PROGRAM PRG_TerminalMapping
VAR
    uiIndexPositionCode : UINT;
END_VAR

METHOD PUBLIC ReadInputs
(*
======================================================================================================================
 Terminal 4 | EL1918
======================================================================================================================
*)
GVL_IO.stInputs.bEmergencyStopChannel1 	:= GVL_EtherCAT.stTerm4_EL1918.iEL1918_Ch1;
GVL_IO.stInputs.bEmergencyStopChannel2 	:= GVL_EtherCAT.stTerm4_EL1918.iEL1918_Ch2;
// Reset is exported by TwinSAFE. Use the validated alias rather than
// reconstructing the operator Reset from a raw safety-terminal channel.
GVL_IO.stInputs.bResetButton 			:= GVL_Safety.bResetButtonPressed;
GVL_IO.stInputs.bMainDoorChannel1 		:= GVL_EtherCAT.stTerm4_EL1918.iEL1918_Ch4;
GVL_IO.stInputs.bMainDoorChannel2 		:= GVL_EtherCAT.stTerm4_EL1918.iEL1918_Ch5;
GVL_IO.stInputs.bMainDoorFeedback 		:= GVL_EtherCAT.stTerm4_EL1918.iEL1918_Ch6;
GVL_IO.stInputs.bMs6FeedbackOk 			:= GVL_EtherCAT.stTerm4_EL1918.iEL1918_Ch7;
GVL_IO.stInputs.bAirExhausted 			:= GVL_EtherCAT.stTerm4_EL1918.iEL1918_Ch8;

(*
======================================================================================================================
 Terminal 5 | EL1918
======================================================================================================================
*)
GVL_IO.stInputs.bTouchButtonLeft 		:= GVL_EtherCAT.stTerm5_EL1918.iEL1918_Ch3;
GVL_IO.stInputs.bTouchButtonRight 		:= GVL_EtherCAT.stTerm5_EL1918.iEL1918_Ch4;
GVL_IO.stInputs.bRightFlapChannel1 		:= GVL_EtherCAT.stTerm5_EL1918.iEL1918_Ch5;
GVL_IO.stInputs.bRightFlapChannel2 		:= GVL_EtherCAT.stTerm5_EL1918.iEL1918_Ch6;
GVL_IO.stInputs.bLeftFlapChannel1 		:= GVL_EtherCAT.stTerm5_EL1918.iEL1918_Ch7;
GVL_IO.stInputs.bLeftFlapChannel2 		:= GVL_EtherCAT.stTerm5_EL1918.iEL1918_Ch8;

(*
======================================================================================================================
 Terminal 7 | EL1809
======================================================================================================================
*)
GVL_IO.stInputs.bStartButton 				:= GVL_EtherCAT.stTerm7_EL1809.iEL1809_Ch1;
GVL_IO.stInputs.bStopButton 				:= NOT GVL_EtherCAT.stTerm7_EL1809.iEL1809_Ch2;
GVL_IO.stInputs.bUp24VPowerSupplyOk 		:= GVL_EtherCAT.stTerm7_EL1809.iEL1809_Ch3;
GVL_IO.stInputs.bUs24VPowerSupplyOk 		:= GVL_EtherCAT.stTerm7_EL1809.iEL1809_Ch4;
GVL_IO.stInputs.b48VPowerSupplyOk 			:= GVL_EtherCAT.stTerm7_EL1809.iEL1809_Ch5;
GVL_IO.stInputs.bIndexPositionSensor1 		:= GVL_EtherCAT.stTerm7_EL1809.iEL1809_Ch6;
GVL_IO.stInputs.bIndexPositionSensor2 		:= GVL_EtherCAT.stTerm7_EL1809.iEL1809_Ch7;
GVL_IO.stInputs.bIndexPositionSensor3 		:= GVL_EtherCAT.stTerm7_EL1809.iEL1809_Ch8;
GVL_IO.stInputs.bIndexCompletedSensor 		:= GVL_EtherCAT.stTerm7_EL1809.iEL1809_Ch9;
GVL_IO.stInputs.bIndexLocked 				:= GVL_EtherCAT.stTerm7_EL1809.iEL1809_Ch10;
GVL_IO.stInputs.bIndexReady 				:= GVL_EtherCAT.stTerm7_EL1809.iEL1809_Ch11;
GVL_IO.stInputs.bLoadingStationEaglePresent := GVL_EtherCAT.stTerm7_EL1809.iEL1809_Ch12;
GVL_IO.stInputs.bRejectChutePartPresent 	:= GVL_EtherCAT.stTerm7_EL1809.iEL1809_Ch13;
GVL_IO.stInputs.bHeatStakeEaglePresent 		:= GVL_EtherCAT.stTerm7_EL1809.iEL1809_Ch14;
GVL_IO.stInputs.bLoadingStationPbupPresent	:= GVL_EtherCAT.stTerm7_EL1809.iEL1809_Ch15;
GVL_IO.stInputs.bPbupMagnetPresent 			:= GVL_EtherCAT.stTerm7_EL1809.iEL1809_Ch16;

(*
======================================================================================================================
 INDEX Position
======================================================================================================================
*)
uiIndexPositionCode := 0;

IF GVL_IO.stInputs.bIndexPositionSensor1 THEN 
	uiIndexPositionCode := uiIndexPositionCode + 1; 
END_IF

IF GVL_IO.stInputs.bIndexPositionSensor2 THEN 
	uiIndexPositionCode := uiIndexPositionCode + 2; 
END_IF

IF GVL_IO.stInputs.bIndexPositionSensor3 THEN 
	uiIndexPositionCode := uiIndexPositionCode + 4; 
END_IF

IF GVL_IO.stInputs.bIndexLocked THEN 
	GVL_IO.stInputs.eIndexPosition := UINT_TO_E_TablePosition(uiIndexPositionCode);
ELSE 
	GVL_IO.stInputs.eIndexPosition := E_TablePosition.Unknown; 
END_IF

(*
======================================================================================================================
 Terminal 8 | EL1809
======================================================================================================================
*)

GVL_IO.stInputs.bStation1SupportRetracted := FALSE; // Retired compatibility field; EL1809 Ch1/Ch2 reserved.
GVL_IO.stInputs.bStation1SupportExtended := FALSE; // Retired compatibility field; EL1809 Ch1/Ch2 reserved.
GVL_IO.stInputs.bStation2SupportRetracted 		:= GVL_EtherCAT.stTerm8_EL1809.iEL1809_Ch3;
GVL_IO.stInputs.bStation2SupportExtended 		:= GVL_EtherCAT.stTerm8_EL1809.iEL1809_Ch4;
GVL_IO.stInputs.bStation3SupportRetracted := FALSE; // Retired compatibility field; raw terminal stays diagnostic-only.
GVL_IO.stInputs.bStation3SupportExtended := FALSE; // Retired compatibility field; raw terminal stays diagnostic-only.
GVL_IO.stInputs.bHorizontalMiniSlideRetracted 	:= GVL_EtherCAT.stTerm8_EL1809.iEL1809_Ch7;
GVL_IO.stInputs.bHorizontalMiniSlideExtended 	:= GVL_EtherCAT.stTerm8_EL1809.iEL1809_Ch8;
GVL_IO.stInputs.bVerticalMiniSlideExtended		:= GVL_EtherCAT.stTerm8_EL1809.iEL1809_Ch9;
GVL_IO.stInputs.bVerticalMiniSlideRetracted 	:= GVL_EtherCAT.stTerm8_EL1809.iEL1809_Ch10;
GVL_IO.stInputs.bIntermediateModuleRetracted := FALSE; // Retired compatibility field; raw terminal stays diagnostic-only.
GVL_IO.stInputs.bIntermediateModuleExtended := FALSE; // Retired compatibility field; raw terminal stays diagnostic-only.
GVL_IO.stInputs.bRotaryGripperOpened 			:= GVL_EtherCAT.stTerm8_EL1809.iEL1809_Ch13;
GVL_IO.stInputs.bRotaryGripperClosed 			:= GVL_EtherCAT.stTerm8_EL1809.iEL1809_Ch14;
GVL_IO.stInputs.bRotaryGripperPick0             := GVL_EtherCAT.stTerm8_EL1809.iEL1809_Ch16;
GVL_IO.stInputs.bRotaryGripperPlace180          := GVL_EtherCAT.stTerm8_EL1809.iEL1809_Ch15;

(*
======================================================================================================================
 Terminal 19 | EL1809
======================================================================================================================
*)

// Provisional operator PBUP presence; move this mapping when the final terminal is assigned.
//GVL_IO.stInputs.bLoadingStationPbupPresent 	:= GVL_EtherCAT.stTerm19_EL1809.iEL1809_Ch1;
GVL_IO.stInputs.bPatchOpticalLeft 			:= GVL_EtherCAT.stTerm19_EL1809.iEL1809_Ch5;
GVL_IO.stInputs.bPatchOpticalRight 			:= GVL_EtherCAT.stTerm19_EL1809.iEL1809_Ch6;
GVL_IO.stInputs.bHeatStakeHeadUp   			:= GVL_EtherCAT.stTerm19_EL1809.iEL1809_Ch7;
GVL_IO.stInputs.bHeatStakeHeadDown 			:= GVL_EtherCAT.stTerm19_EL1809.iEL1809_Ch8;
GVL_IO.stInputs.bMembraneTransferRetracted 	:= GVL_EtherCAT.stTerm19_EL1809.iEL1809_Ch9;
GVL_IO.stInputs.bMembraneTransferExtended 	:= GVL_EtherCAT.stTerm19_EL1809.iEL1809_Ch10;
GVL_IO.stInputs.bMiddleRockerDown 			:= GVL_EtherCAT.stTerm19_EL1809.iEL1809_Ch11;
GVL_IO.stInputs.bMiddleRockerUp 			:= GVL_EtherCAT.stTerm19_EL1809.iEL1809_Ch12;
GVL_IO.stInputs.bBottomRockerDown 			:= GVL_EtherCAT.stTerm19_EL1809.iEL1809_Ch13;
GVL_IO.stInputs.bBottomRockerUp 			:= GVL_EtherCAT.stTerm19_EL1809.iEL1809_Ch14;
GVL_IO.stInputs.bTopRockerDown 				:= GVL_EtherCAT.stTerm19_EL1809.iEL1809_Ch15;
GVL_IO.stInputs.bTopRockerUp 				:= GVL_EtherCAT.stTerm19_EL1809.iEL1809_Ch16;

(*
======================================================================================================================
 Terminal 11 | EL3058
======================================================================================================================
*)
GVL_IO.stInputs.uiMainAirPressureRaw 		 := GVL_EtherCAT.stTerm11_EL3058.iEL3058_Ch1;
GVL_IO.stInputs.uiPressureRegulatorActualRaw := GVL_EtherCAT.stTerm11_EL3058.iEL3058_Ch2;

(*
======================================================================================================================
 Terminal 20 | EL3314-0092 | Heat Stake Thermocouples
======================================================================================================================
*)
GVL_IO.stInputs.diHeatStakeTc1Raw := GVL_EtherCAT.stTerm21_EL3314.iEL3314_Ch1;
GVL_IO.stInputs.diHeatStakeTc2Raw := GVL_EtherCAT.stTerm21_EL3314.iEL3314_Ch2;
GVL_IO.stInputs.diHeatStakeTc3Raw := GVL_EtherCAT.stTerm21_EL3314.iEL3314_Ch3;

(*
======================================================================================================================
 SAFETY ALIAS Inputs
======================================================================================================================
*)
GVL_IO.stInputs.bSafetyOk 				:= GVL_Safety.bSafetyOk;
GVL_IO.stInputs.bTwoHandsSafe 			:= GVL_Safety.bTwoHandSafe;
GVL_IO.stInputs.bMainDoorClosed 		:= GVL_Safety.bMainDoorClosed;
GVL_IO.stInputs.bMainDoorLocked 		:= GVL_Safety.bMainDoorLocked;
GVL_IO.stInputs.bMainDoorUnsafe 		:= GVL_Safety.bMainDoorUnSafe;
GVL_IO.stInputs.bMainDoorDiagnosticOk 	:= GVL_Safety.bMainDoorDiagnosticOk;
END_METHOD

METHOD PUBLIC WriteOutputs
(*
======================================================================================================================
 SAFETY Alias Outputs
======================================================================================================================
*)
GVL_Safety.bSafetyRunRequest 					:= GVL_IO.stOutputs.bSafetyRunRequest;
GVL_Safety.bSafetyResetRequest 					:= GVL_IO.stOutputs.bSafetyResetRequest;
GVL_Safety.bSafetyErrorAcknowledgementRequest 	:= GVL_IO.stOutputs.bSafetyErrorAcknowledgementRequest;
GVL_Safety.bAirSupplyEnableRequest 				:= GVL_IO.stOutputs.bAirSupplyEnable;
GVL_Safety.bMainDoorLockRequest 				:= GVL_IO.stOutputs.bMainDoorLockRequest;

(*
======================================================================================================================
 Terminal 9 | EL2809
======================================================================================================================
*)
GVL_EtherCAT.stTerm9_EL2809.iEL2809_Ch1 := GVL_IO.stOutputs.bLedStart;
GVL_EtherCAT.stTerm9_EL2809.iEL2809_Ch2 := GVL_IO.stOutputs.bLedReset;

// Validated physical status-light mapping:
// Ch3 = RED status indicator (driven from machine FAIL)
// Ch4 = GREEN status indicator (driven from machine PASS)
GVL_EtherCAT.stTerm9_EL2809.iEL2809_Ch3 := GVL_IO.stOutputs.bStatusIndicatorRed;
GVL_EtherCAT.stTerm9_EL2809.iEL2809_Ch4 := GVL_IO.stOutputs.bStatusIndicatorGreen;

// Ch5 = internal cabinet/machine light
// Ch6 = operator/nest light
GVL_EtherCAT.stTerm9_EL2809.iEL2809_Ch5 := GVL_IO.stOutputs.bInternalLight;
GVL_EtherCAT.stTerm9_EL2809.iEL2809_Ch6 := GVL_IO.stOutputs.bNestLight;
// Monostable Heat Stake valve: TRUE = UP, FALSE = DOWN.
GVL_EtherCAT.stTerm9_EL2809.iEL2809_Ch7 := GVL_IO.stOutputs.bHeatStakeHeadUp;

(*
======================================================================================================================
 Terminal 13 | EL2502 | Heat Stake PWM Outputs
======================================================================================================================
*)
// IMPORTANT - VALIDATED PHYSICAL MAPPING.
// The heater channels are intentionally crossed relative to logical Heater 1 / Heater 2.
//
// EL2502 Ch1 physically drives logical Heater 2.
// EL2502 Ch2 physically drives logical Heater 1.
GVL_EtherCAT.stTerm13_EL2502.iEL2502_Ch1 := GVL_IO.stOutputs.uiHeatStakePwm2Raw;
GVL_EtherCAT.stTerm13_EL2502.iEL2502_Ch2 := GVL_IO.stOutputs.uiHeatStakePwm1Raw;

(*
======================================================================================================================
 Terminal 21 | EL4028 | VEAB Heat Stake Down Pressure
======================================================================================================================
*)
GVL_EtherCAT.stTerm20_EL4022.iEL4028_Ch1 := GVL_IO.stOutputs.iHeatStakePressureRaw;

(*
======================================================================================================================
 BOX 1 | Festo VABX EtherCAT manifold - Module 2
======================================================================================================================
*)

// Module2.Coil0 = Index Table A - rotate index
// Module2.Coil1 = Index Table B - return index cylinder to home
// Module2.Coil2 = RESERVED - removed Patch nest support UP
// Module2.Coil3 = RESERVED - removed Patch nest support DOWN
// Module2.Coil4 = Support UP   - Heat Stake Station
// Module2.Coil5 = Support DOWN - Heat Stake Station
// Module2.Coil6 = Support UP   - Vision Station
// Module2.Coil7 = Support DOWN - Vision Station
//
// Application naming:
// UP   = Extend
// DOWN = Retract
GVL_EtherCAT.stFestoModule2_VABX.bCoil0 := GVL_IO.stOutputs.bIndexRotatePortA;
GVL_EtherCAT.stFestoModule2_VABX.bCoil1 := GVL_IO.stOutputs.bIndexStopPortB;

GVL_EtherCAT.stFestoModule2_VABX.bCoil2 := FALSE; // Removed Patch nest support; keep valve OFF.
GVL_EtherCAT.stFestoModule2_VABX.bCoil3 := FALSE; // Reserved, not reassigned.

GVL_EtherCAT.stFestoModule2_VABX.bCoil4 := GVL_IO.stOutputs.bStation2SupportExtend;
GVL_EtherCAT.stFestoModule2_VABX.bCoil5 := GVL_IO.stOutputs.bStation2SupportRetract;

GVL_EtherCAT.stFestoModule2_VABX.bCoil6 := FALSE; // Removed Vision hardware: never energise.
GVL_EtherCAT.stFestoModule2_VABX.bCoil7 := FALSE; // Removed Vision hardware: never energise.

(*
======================================================================================================================
 BOX 1 | Festo VABX EtherCAT manifold - Module 3 | Vision Flipping
======================================================================================================================
*)
// Mapping confirmed from the commissioned GVL_EtherCAT / manifold layout.
// Coil0 = Horizontal slide BACK
// Coil1 = Horizontal slide FRONT
// Coil2 = Vertical cylinder UP
// Coil3 = Vertical cylinder DOWN
// Coil4 = Vertical cylinder limit OFF
// Coil5 = Vertical cylinder limit ON
// Coil6 = Grip CLOSE
// Coil7 = Grip OPEN
GVL_EtherCAT.stFestoModule3_VABX.bCoil0 := GVL_IO.stOutputs.bVisionHorizontalBack;
GVL_EtherCAT.stFestoModule3_VABX.bCoil1 := GVL_IO.stOutputs.bVisionHorizontalFront;
GVL_EtherCAT.stFestoModule3_VABX.bCoil2 := GVL_IO.stOutputs.bVisionVerticalUp;
GVL_EtherCAT.stFestoModule3_VABX.bCoil3 := GVL_IO.stOutputs.bVisionVerticalDown;
GVL_EtherCAT.stFestoModule3_VABX.bCoil4 := FALSE; // Removed Vision hardware: never energise.
GVL_EtherCAT.stFestoModule3_VABX.bCoil5 := FALSE; // Removed Vision hardware: never energise.
GVL_EtherCAT.stFestoModule3_VABX.bCoil6 := GVL_IO.stOutputs.bVisionGripOpen;
GVL_EtherCAT.stFestoModule3_VABX.bCoil7 := GVL_IO.stOutputs.bVisionGripClose;
(*
======================================================================================================================
 BOX 1 | Festo VABX EtherCAT manifold - Module 4 | Heat Stake Head
======================================================================================================================
*)
// Mapping confirmed from the commissioned GVL_EtherCAT / manifold layout.
// Coil0 = Vision gripper rotation 0Â° / PICK
// Coil1 = Vision gripper rotation 180Â° / PLACE
// Coil2 = Patch dispenser AIR
// Coil3 = Heat Stake head UNLOCK
// Coil4 = retired head DOWN output (always OFF)
// Coil5 = continuous pilot supply for the external head valve
// Coil6 = Patch vertical support DOWN
// Coil7 = Patch vertical support UP

GVL_EtherCAT.stFestoModule4_VABX.bCoil0 := GVL_IO.stOutputs.bVisionRotate0;
GVL_EtherCAT.stFestoModule4_VABX.bCoil1 := GVL_IO.stOutputs.bVisionRotate180;
GVL_EtherCAT.stFestoModule4_VABX.bCoil2 := GVL_IO.stOutputs.bPatchDispenserAir;
GVL_EtherCAT.stFestoModule4_VABX.bCoil3 := GVL_IO.stOutputs.bHeatStakeHeadUnlock;
GVL_EtherCAT.stFestoModule4_VABX.bCoil4 := FALSE; // Retired direction output.
GVL_EtherCAT.stFestoModule4_VABX.bCoil5 := TRUE; // Continuous pilot supply; reservoir supports retraction.
GVL_EtherCAT.stFestoModule4_VABX.bCoil6 := GVL_IO.stOutputs.bPatchVerticalDown;
GVL_EtherCAT.stFestoModule4_VABX.bCoil7 := GVL_IO.stOutputs.bPatchVerticalUp;
END_METHOD

END_PROGRAM

(* stored: Version 1.1.0.1, ProductVersion 3.1.4026.18
   POU PRG_TerminalMapping: Id {238243cb-7891-4569-b868-8787a9e2c958}, SpecialFunc None
   Method ReadInputs: Id {dd42962b-99a1-4f07-bcc4-f10d6e3158eb}
   Method WriteOutputs: Id {d5ba67cb-64f8-4d86-bcb1-1981d0b6759b} *)
